% RSLogix 500 project CE Autolavado.RSS, saved by version 8.40.00.08 %
PROJECT "UNTITLED"    % processor: MicroLogix 1200 %

PROGRAM FILES
  LAD 2   14 rungs

DATA FILES
  O0 OUTPUT  4 elements
  I1 INPUT  4 elements
  S2 STATUS  66 elements
  B3 BINARY  1 elements
  T4 TIMER  3 elements
  C5 COUNTER  1 elements
  R6 CONTROL  1 elements
  N7 INTEGER  1 elements
  F8 FLOAT  1 elements

LADDER 2
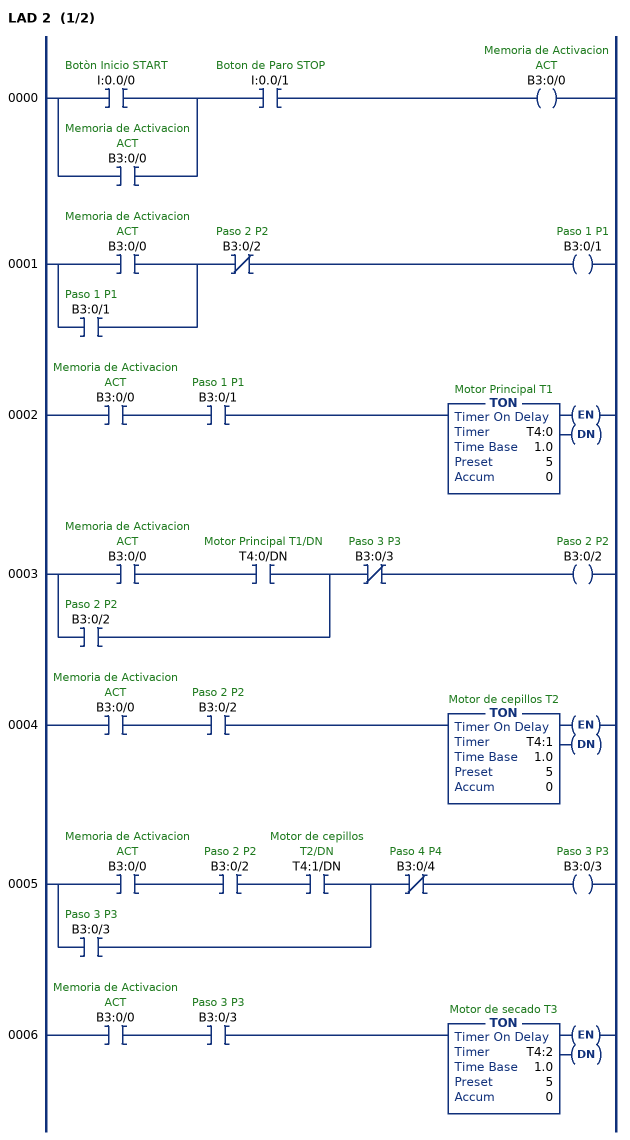
% Rung: 0 %
SOR BST XIC I:0.0/0 NXB XIC B3:0/0 BND XIC I:0.0/1 OTE B3:0/0 EOR
%   I:0.0/0  START  "Botòn Inicio" %
%   B3:0/0  ACT  "Memoria de Activacion" %
%   I:0.0/1  STOP  "Boton de Paro" %
% Rung: 1 %
SOR BST XIC B3:0/0 NXB XIC B3:0/1 BND XIO B3:0/2 OTE B3:0/1 EOR
%   B3:0/0  ACT  "Memoria de Activacion" %
%   B3:0/1  P1  "Paso 1" %
%   B3:0/2  P2  "Paso 2" %
% Rung: 2 %
SOR XIC B3:0/0 XIC B3:0/1 TON T4:0 1.0 5 0 EOR
%   B3:0/0  ACT  "Memoria de Activacion" %
%   B3:0/1  P1  "Paso 1" %
%   T4:0  T1  "Motor Principal" %
% Rung: 3 %
SOR BST XIC B3:0/0 XIC T4:0/DN NXB XIC B3:0/2 BND XIO B3:0/3 OTE B3:0/2 EOR
%   B3:0/0  ACT  "Memoria de Activacion" %
%   T4:0  T1  "Motor Principal" %
%   B3:0/2  P2  "Paso 2" %
%   B3:0/3  P3  "Paso 3" %
% Rung: 4 %
SOR XIC B3:0/0 XIC B3:0/2 TON T4:1 1.0 5 0 EOR
%   B3:0/0  ACT  "Memoria de Activacion" %
%   B3:0/2  P2  "Paso 2" %
%   T4:1  T2  "Motor de cepillos" %
% Rung: 5 %
SOR BST XIC B3:0/0 XIC B3:0/2 XIC T4:1/DN NXB XIC B3:0/3 BND XIO B3:0/4 OTE B3:0/3 EOR
%   B3:0/0  ACT  "Memoria de Activacion" %
%   B3:0/2  P2  "Paso 2" %
%   T4:1  T2  "Motor de cepillos" %
%   B3:0/3  P3  "Paso 3" %
%   B3:0/4  P4  "Paso 4" %
% Rung: 6 %
SOR XIC B3:0/0 XIC B3:0/3 TON T4:2 1.0 5 0 EOR
%   B3:0/0  ACT  "Memoria de Activacion" %
%   B3:0/3  P3  "Paso 3" %
%   T4:2  T3  "Motor de secado" %

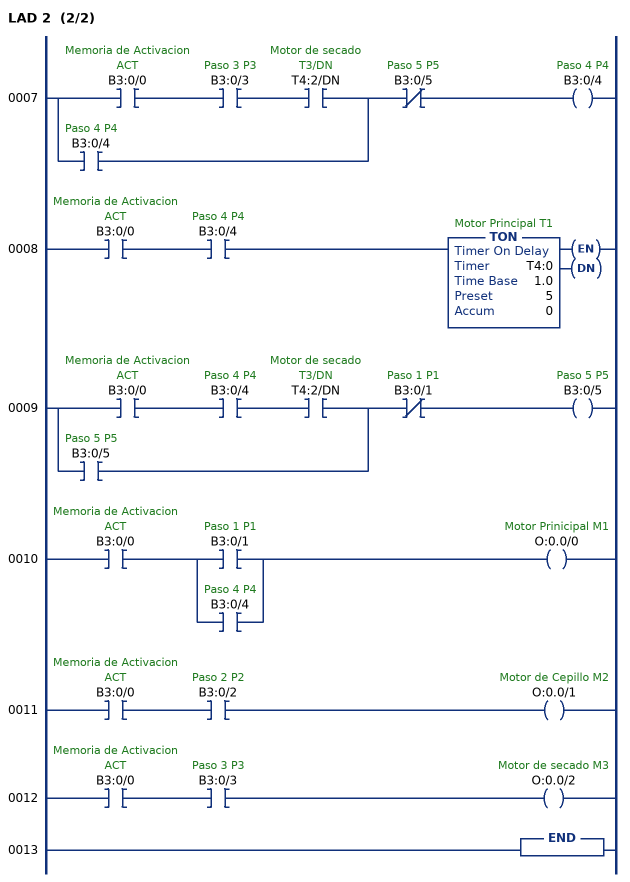
% Rung: 7 %
SOR BST XIC B3:0/0 XIC B3:0/3 XIC T4:2/DN NXB XIC B3:0/4 BND XIO B3:0/5 OTE B3:0/4 EOR
%   B3:0/0  ACT  "Memoria de Activacion" %
%   B3:0/3  P3  "Paso 3" %
%   T4:2  T3  "Motor de secado" %
%   B3:0/4  P4  "Paso 4" %
%   B3:0/5  P5  "Paso 5" %
% Rung: 8 %
SOR XIC B3:0/0 XIC B3:0/4 TON T4:0 1.0 5 0 EOR
%   B3:0/0  ACT  "Memoria de Activacion" %
%   B3:0/4  P4  "Paso 4" %
%   T4:0  T1  "Motor Principal" %
% Rung: 9 %
SOR BST XIC B3:0/0 XIC B3:0/4 XIC T4:2/DN NXB XIC B3:0/5 BND XIO B3:0/1 OTE B3:0/5 EOR
%   B3:0/0  ACT  "Memoria de Activacion" %
%   B3:0/4  P4  "Paso 4" %
%   T4:2  T3  "Motor de secado" %
%   B3:0/5  P5  "Paso 5" %
%   B3:0/1  P1  "Paso 1" %
% Rung: 10 %
SOR XIC B3:0/0 BST XIC B3:0/1 NXB XIC B3:0/4 BND OTE O:0.0/0 EOR
%   B3:0/0  ACT  "Memoria de Activacion" %
%   B3:0/1  P1  "Paso 1" %
%   B3:0/4  P4  "Paso 4" %
%   O:0.0/0  M1  "Motor Prinicipal" %
% Rung: 11 %
SOR XIC B3:0/0 XIC B3:0/2 OTE O:0.0/1 EOR
%   B3:0/0  ACT  "Memoria de Activacion" %
%   B3:0/2  P2  "Paso 2" %
%   O:0.0/1  M2  "Motor de Cepillo" %
% Rung: 12 %
SOR XIC B3:0/0 XIC B3:0/3 OTE O:0.0/2 EOR
%   B3:0/0  ACT  "Memoria de Activacion" %
%   B3:0/3  P3  "Paso 3" %
%   O:0.0/2  M3  "Motor de secado" %
% Rung: 13 %
SOR END EOR

DATA TABLE (non-zero values as saved)
DATA T4
% .PRE .ACC %
% T4:0 % 5 0
% T4:1 % 5 0
% T4:2 % 5 0
